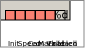
VISUALIZATION _VISU_MarkDetection_Trigger  // 85x48
VAR_IN_OUT
	mInst : FB_MarkDetection;
END_VAR
    RoundedRectangle (0,0 70x20), tooltip "Trigger Armed", colour toggle: mInst.bTriggerArmed
    RoundedRectangle (15,10 10x10), tooltip "Speed valid", colour toggle: mInst.bSpeedValid
    RoundedRectangle (25,10 10x10), tooltip "Cam valid", colour toggle: mInst.bCamValid
    RoundedRectangle (35,10 10x10), tooltip "marks valid", colour toggle: mInst.bMarkValid
    RoundedRectangle (5,10 10x10), tooltip "Init ok", colour toggle: mInst.bInitOk
    Rectangle (0,0 70x10), tooltip "Trigger active"
    RoundedRectangle (55,10 10x10), "%d", tooltip "e state", text variable: mInst.nMarkSelection
    RoundedRectangle (45,10 10x10), tooltip "(Hw)Enable", colour toggle: mInst.bEnable
    Rectangle (-12,38 45x10), angle 90, "Init"
    Rectangle (-2,38 45x10), angle 90, "Speed"
    Rectangle (8,38 45x10), angle 90, "Cam Valid"
    Rectangle (18,38 45x10), angle 90, "Mark teach"
    Rectangle (28,38 45x10), angle 90, "Enabled"
END_VISUALIZATION

(* stored: Version 1.1.0.1, ProductVersion 3.1.4024.11
   Visu _VISU_MarkDetection_Trigger: Id {57ea54a9-6327-495f-a500-87f69f5bc301} *)
